Staubli VAL3: IoWriteRequestMsg.dtx

public Body body
  [0]
    num nData[28]
public Header header
  [0]
    num nMsgType
    num nCommType
    num nReplyCode
    num nData[9]
public Prefix prefix
  [0]
    num nLength
    num nData[4]
public IoWriteRequest ioWriteRequest
  [0]
    num nCount
    num nType
    num nIndex
    num nValue
